// TIA Portal V19 export
DATA_BLOCK "AO SCALING DB"   // DB134
{ S7_Optimized_Access := 'FALSE' }
   VAR
      SET : Struct
         "VFD P-501A" : Real;
         "VFD P-501B" : Real;
         "VFD P-501C" : Real;
      END_STRUCT;
      MIN : Struct
         "VFD P-501A" : Real;
         "VFD P-501B" : Real;
         "VFD P-501C" : Real;
      END_STRUCT;
      MAX : Struct
         "VFD P-501A" { S7_SetPoint := 'True'} : Real := 50.0;
         "VFD P-501B" { S7_SetPoint := 'True'} : Real := 50.0;
         "VFD P-501C" { S7_SetPoint := 'True'} : Real := 50.0;
      END_STRUCT;
      PV : Struct
         "VFD P-501A" : Real;
         "VFD P-501B" : Real;
         "VFD P-501C" : Real;
      END_STRUCT;
   END_VAR
BEGIN
END_DATA_BLOCK
